FUNCTION_BLOCK ModeControl_Mockup EXTENDS ModeControl
VAR
	{attribute 'hide'}
	_IsChangeModeInvoked : BOOL;
	{attribute 'hide'}
	_LastRequestedMode : DINT;
	{attribute 'hide'}
	_IsExecuting : BOOL;
END_VAR

// Override the ChangeMode method to add mockup tracking
METHOD ChangeMode
VAR_INPUT
	RequestedMode : DINT;
END_VAR
_IsChangeModeInvoked := TRUE;
_LastRequestedMode	 := RequestedMode;
_IsExecuting		 := TRUE;

// Call the base implementation
SUPER^.ChangeMode(RequestedMode);
END_METHOD

// Method to complete/reset execution state
METHOD Complete
_IsExecuting		 := FALSE;
_IsChangeModeInvoked := FALSE;
_LastRequestedMode	 := 0;
END_METHOD

// Mockup specific method to simulate execution state
METHOD Executing
_IsExecuting := TRUE;
END_METHOD

// Additional method to check if ChangeMode was called
METHOD IsExecuting : BOOL
IsExecuting := _IsExecuting;
END_METHOD

END_FUNCTION_BLOCK

(* stored: Version 1.1.0.1, ProductVersion 3.1.4026.18
   POU ModeControl_Mockup: Id {ffe7bd8f-32c4-481d-b9b9-d57410f3e5a6}, SpecialFunc None
   Method ChangeMode: Id {56cb1f75-fe1f-4b3f-afe7-3774cfd68893}
   Method Complete: Id {487118ad-ddc0-41a9-8bc0-335f2c763b4a}
   Method Executing: Id {511bba75-592d-458c-9ff7-bf9a64a65085}
   Method IsExecuting: Id {78a1caf7-e36d-4b5c-a083-483ce54243eb} *)
